// TIA Portal V19 export
TYPE "LEXCHANGETRAY_typeRoller_toLogisticsDeliver"
// stored: Access Published
   STRUCT
      feedback : "LEXCHANGETRAY_typeRoller_toLogisticsFeedback";
      req { S7_SetPoint := 'True'} : "LEXCHANGETRAY_typeRoller_toLogisticsReq";
   END_STRUCT;
END_TYPE
